Fanuc KAREL source: prog_x.kl

PROGRAM prog_x
%ALPHABETIZE
%COMMENT = ''
%NOBUSYLAMP
%NOLOCKGROUP
%NOPAUSE = COMMAND + TPENABLE + ERROR

%include lib_a\a.klt

%mode push
%mode string QQQ "`" "`" "\\"
%define t_arr2d(y,x,n,t) `TYPE
  #3_0 = ARRAY[x] OF #4
  #3_1 = ARRAY[y] OF #3_0`
%define arrx(n) %eval #1_0
%define arry(n) %eval #1_1
%mode pop

t_arr2d(5,10,rarr,REAL)

VAR
  i,j     : INTEGER
  rows    : arrx(rarr)
  a_2d    : arry(rarr)

%include lib_a\a.klh

BEGIN
  --run subroutines from lib_a
	a_clrscr
	a_do_smthng(1)

  --test type macro from ktransw-macros
  FOR i=1 TO ARRAY_LEN(a_2d) DO
    FOR j=1 TO ARRAY_LEN(rows) DO
      rows[j] = j*i
    ENDFOR

    a_2d[i] = rows
  ENDFOR

END prog_x
